FUNCTION_BLOCK FB_Heating
VAR_INPUT
	bInput			:	BOOL;
	bInputOverwrite	:	BOOL;
END_VAR
VAR_OUTPUT
	bOut			:	BOOL;
END_VAR
VAR
END_VAR

IF bInputOverwrite THEN
	bOut := TRUE;
ELSE
	bOut := bInput;
END_IF

END_FUNCTION_BLOCK

(* stored: Version 1.1.0.1, ProductVersion 3.1.4024.4
   POU FB_Heating: Id {9baa2ebe-d006-4adc-9e0a-95958572b8cd}, SpecialFunc None *)
